(* Visualisation Visualizace
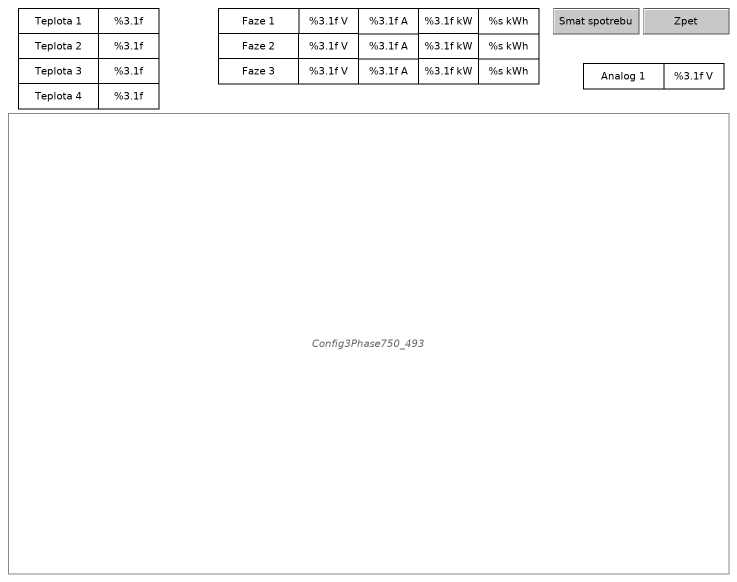
rectangle at (30,35)-(111,61): text "Teplota 1"
rectangle at (30,60)-(111,86): text "Teplota 2"
rectangle at (30,85)-(111,111): text "Teplota 3"
rectangle at (30,110)-(111,136): text "Teplota 4"
rectangle at (110,35)-(171,61): text "%3.1f"; shows .Teplota_1/10.0
rectangle at (110,60)-(171,86): text "%3.1f"; shows .Teplota_2/10.0
rectangle at (110,85)-(171,111): text "%3.1f"; shows .Teplota_3/10.0
rectangle at (110,110)-(171,136): text "%3.1f"; shows .Teplota_4/10.0
rectangle at (675,90)-(736,116): text "%3.1f V"; shows .Analog_1/3276.4
rectangle at (595,90)-(676,116): text "Analog 1"
rectangle at (310,35)-(371,61): text "%3.1f V"; shows TriFaze.arNapeti[1]
rectangle at (230,35)-(311,61): text "Faze 1"
rectangle at (230,60)-(311,86): text "Faze 2"
rectangle at (230,85)-(311,111): text "Faze 3"
embedded screen at (20,140)-(741,601): Config3Phase750_493
rectangle at (310,60)-(371,86): text "%3.1f V"; shows TriFaze.arNapeti[2]
rectangle at (310,85)-(371,111): text "%3.1f V"; shows TriFaze.arNapeti[3]
rectangle at (370,85)-(431,111): text "%3.1f A"; shows TriFaze.arProud[3]
rectangle at (370,60)-(431,86): text "%3.1f A"; shows TriFaze.arProud[2]
rectangle at (370,35)-(431,61): text "%3.1f A"; shows TriFaze.arProud[1]
rectangle at (430,35)-(491,61): text "%3.1f kW"; shows TriFaze.arVykon[1]
rectangle at (430,60)-(491,86): text "%3.1f kW"; shows TriFaze.arVykon[2]
rectangle at (430,85)-(491,111): text "%3.1f kW"; shows TriFaze.arVykon[3]
rectangle at (490,85)-(551,111): text "%s kWh"; shows TriFaze.adwSpotreba[3]
rectangle at (490,60)-(551,86): text "%s kWh"; shows TriFaze.adwSpotreba[2]
rectangle at (490,35)-(551,61): text "%s kWh"; shows TriFaze.adwSpotreba[1]
button at (565,35)-(651,61): text "Smat spotrebu"; taps TriFaze.SmazL1
button at (655,35)-(741,61): text "Zpet"; opens PLC_VISU
*)
